(* PLC project mtcs_cover, Institute of Astronomy Onto 0.0.1 *)
(* stored: creationDateTime 2025-01-10T14:32:38.371541, modificationDateTime 2025-01-10T14:32:38.371541 *)

TYPE CoverApertureProcedureStates : (IDLE := 0, ABORTED := 1, PREPARE_PROCESS := 2, ENABLING_RELAYS := 3, ENABLING_MOTORS := 4, ENABLING_MAGNETS := 5, DISABLING_RELAYS := 6, DISABLING_MOTORS := 7, DISABLING_MAGNETS := 8, OPENING_TOP_PANELS := 9, OPENING_BOTH_PANELS := 10, CLOSING_BOTTOM_PANELS := 11, CLOSING_BOTH_PANELS := 12, ERROR := 13, RESETTING := 14, ABORTING := 15);
END_TYPE

TYPE CoverParts : STRUCT
  top : CoverPanelSet;  (* TOP panels *)
  bottom : CoverPanelSet;  (* BOTTOM panels *)
  io : CoverIO;  (* I/O modules *)
  apertureProcedure : CoverApertureProcedure;  (* The closing/opening/... procedure *)
  configManager : ConfigManager;  (* The config manager (to load/save/activate configuration data) *)
END_STRUCT;
END_TYPE

TYPE CoverPanelSetParts : STRUCT
  p1 : CoverPanel;  (* Panel 1 *)
  p2 : CoverPanel;  (* Panel 2 *)
  p3 : CoverPanel;  (* Panel 3 *)
  p4 : CoverPanel;  (* Panel 4 *)
  magnetsRelay : SimpleRelay;  (* Relay for the magnets of this panelset *)
END_STRUCT;
END_TYPE

TYPE CoverPanelParts : STRUCT
  axis : AngularAxis;  (* NC Axis *)
  motorRelay : SimpleRelay;  (* Relay for the motor *)
END_STRUCT;
END_TYPE

TYPE CoverIOParts : STRUCT
  coupler : EtherCatDevice;  (* Coupler *)
  slot1 : EtherCatDevice;  (* Slot 1 *)
  slot2 : EtherCatDevice;  (* Slot 2 *)
  slot3 : EtherCatDevice;  (* Slot 3 *)
  slot4 : EtherCatDevice;  (* Slot 4 *)
  slot5 : EtherCatDevice;  (* Slot 5 *)
  slot6 : EtherCatDevice;  (* Slot 6 *)
  slot7 : EtherCatDevice;  (* Slot 7 *)
  slot8 : EtherCatDevice;  (* Slot 8 *)
  slot9 : EtherCatDevice;  (* Slot 9 *)
  slot10 : EtherCatDevice;  (* Slot 10 *)
  slot11 : EtherCatDevice;  (* Slot 11 *)
  slot12 : EtherCatDevice;  (* Slot 12 *)
  slot13 : EtherCatDevice;  (* Slot 13 *)
END_STRUCT;
END_TYPE

TYPE CoverProcesses : STRUCT
  initialize : Process;  (* Start initializing *)
  lock : Process;  (* Lock the cover *)
  unlock : Process;  (* Unlock the cover *)
  reset : Process;  (* Reset any errors *)
  changeOperatingState : ChangeOperatingStateProcess;  (* Change the operating state (e.g. AUTO, MANUAL, ...) *)
  open : Process;  (* Start opening the cover (only enabled in AUTO mode!) *)
  close : Process;  (* Start closing the cover (only enabled in AUTO mode!) *)
  forceOpen : Process;  (* Start opening the cover EVEN IF WE'RE IN THE UNSAFE REGION *)
  forceClose : Process;  (* Start closing the cover EVEN IF WE'RE IN THE UNSAFE REGION *)
  abort : Process;  (* Abort opening/closing the cover (only enabled in AUTO mode!) *)
END_STRUCT;
END_TYPE

TYPE CoverPanelSetProcesses : STRUCT
  reset : Process;  (* Reset any errors *)
END_STRUCT;
END_TYPE

TYPE CoverPanelProcesses : STRUCT
  startOpening : Process;  (* Start opening the panel *)
  startClosing : Process;  (* Start closing the panel *)
END_STRUCT;
END_TYPE

TYPE CoverStatuses : STRUCT
  initializationStatus : InitializationStatus;
  apertureStatus : ApertureStatus;
  healthStatus : HealthStatus;
  busyStatus : BusyStatus;
  operatingStatus : OperatingStatus;
END_STRUCT;
END_TYPE

TYPE CoverApertureProcedureStatuses : STRUCT
  busyStatus : BusyStatus;  (* Is the CoverApertureProcedure in a busy state? *)
  healthStatus : HealthStatus;  (* Is the CoverApertureProcedure in a healthy state? *)
END_STRUCT;
END_TYPE

TYPE CoverPanelSetStatuses : STRUCT
  apertureStatus : ApertureStatus;
  healthStatus : HealthStatus;
  busyStatus : BusyStatus;
END_STRUCT;
END_TYPE

TYPE CoverPanelStatuses : STRUCT
  busyStatus : BusyStatus;  (* Is the panel in a busy state? *)
  apertureStatus : ApertureStatus;  (* Is the panel open or closed? *)
  healthStatus : HealthStatus;  (* Is the panel in a healthy state? *)
  openingStatus : OpeningStatus;  (* Is the panel opening or closing or standing still? *)
END_STRUCT;
END_TYPE

TYPE CoverIOStatuses : STRUCT
  healthStatus : HealthStatus;  (* Is the I/O in a healthy state? *)
END_STRUCT;
END_TYPE

TYPE CoverConfig : STRUCT
  top : CoverPanelSetConfig;  (* The config of the top panel set *)
  bottom : CoverPanelSetConfig;  (* The config of the bottom panel set *)
  openingVelocity : LREAL := 20.0;  (* The opening velocity of the panels in degrees per second (always positive!) *)
  closingVelocity : LREAL := 20.0;  (* The closing velocity of the panels in degrees per second (always positive!) *)
  magnetRemanentTime : LREAL := 3.0;  (* How many seconds should be waited after disabling a magnet, before a panel may move? *)
  targetDistanceBetweenPanelSets : LREAL;  (* The minimum distance in degrees between both panelsets *)
  minDistanceBetweenPanelSets : LREAL;  (* The minimum distance in degrees between both panelsets *)
  unsafeRangeMinElevation : LREAL;  (* The minimum elevation of the unsafe range *)
  unsafeRangeMinAzimuth : LREAL;  (* The minimum azimuth of the unsafe range *)
  unsafeRangeMaxAzimuth : LREAL;  (* The maximum azimuth of the unsafe range *)
END_STRUCT;
END_TYPE

TYPE CoverPanelSetConfig : STRUCT
  p1 : CoverPanelConfig;  (* The config of the first panel of this set *)
  p2 : CoverPanelConfig;  (* The config of the second panel of this set *)
  p3 : CoverPanelConfig;  (* The config of the third panel of this set *)
  p4 : CoverPanelConfig;  (* The config of the fourth panel of this set *)
  name : STRING;  (* The name of the panel set *)
END_STRUCT;
END_TYPE

TYPE CoverPanelConfig : STRUCT
  closedPosition : LREAL;  (* The closed position of the panel in degrees *)
  openPosition : LREAL;  (* The open position of the panel in degrees *)
  openTolerance : LREAL;  (* The tolerance for opening, in degrees *)
  closedTolerance : LREAL;  (* The tolerance for closing, in degrees *)
  standstillTolerance : LREAL;  (* Tolerance in degrees per second: if smaller than ABS(this value), then the cover panel is considered to be standing still *)
  name : STRING;  (* The name of the panel *)
  offset : LREAL;  (* The offset of the panel w.r.t. north *)
END_STRUCT;
END_TYPE

FUNCTION_BLOCK SM_Cover
  VAR_INPUT
    {attribute 'OPC.UA.DA' := '1'}
    {attribute 'OPC.UA.DA.Access' := '1'}
    editableConfig : CoverConfig;  (* Editable configuration of the cover *)
  END_VAR
  VAR_OUTPUT
    {attribute 'OPC.UA.DA' := '1'}
    {attribute 'OPC.UA.DA.Access' := '1'}
    actualStatus : STRING;  (* Current status description *)
    previousStatus : STRING;  (* Previous status description *)
    {attribute 'OPC.UA.DA' := '1'}
    {attribute 'OPC.UA.DA.Access' := '1'}
    config : CoverConfig;  (* Active configuration of the cover *)
    {attribute 'OPC.UA.DA' := '1'}
    {attribute 'OPC.UA.DA.Access' := '1'}
    currentMeasurement : CurrentMeasurement;  (* The current measurement of the selected panels *)
    {attribute 'OPC.UA.DA' := '1'}
    {attribute 'OPC.UA.DA.Access' := '1'}
    safeToOpenOrClose : BOOL;  (* True if safe to open or close! *)
    statuses : CoverStatuses;  (* Statuses of the state machine *)
    parts : CoverParts;  (* Parts of the state machine *)
    processes : CoverProcesses;  (* Processes of the state machine *)
  END_VAR
  VAR_IN_OUT
    {attribute 'OPC.UA.DA' := '0'}
    operatorStatus : OperatorStatus;
    {attribute 'OPC.UA.DA' := '0'}
    aziPos : AngularPosition;  (* Actual azimuth position of the telescope *)
    {attribute 'OPC.UA.DA' := '0'}
    elePos : AngularPosition;  (* Actual elevation position of the telescope *)
  END_VAR

            currentMeasurement();
parts.top(
    initializationStatus := statuses.initializationStatus,
    operatorStatus := operatorStatus,
    operatingStatus := statuses.operatingStatus,
    config := config.top,
    coverConfig := config);
parts.bottom(
    initializationStatus := statuses.initializationStatus,
    operatorStatus := operatorStatus,
    operatingStatus := statuses.operatingStatus,
    config := config.bottom,
    coverConfig := config);
parts.io();
parts.apertureProcedure(
    top := parts.top,
    bottom := parts.bottom,
    coverConfig := config);
parts.configManager( isEnabled := operatorStatus.tech AND statuses.initializationStatus.initialized );
statuses.initializationStatus();
statuses.apertureStatus(
    isOpen := parts.top.statuses.apertureStatus.open AND parts.bottom.statuses.apertureStatus.open,
    isClosed := parts.top.statuses.apertureStatus.closed AND parts.bottom.statuses.apertureStatus.closed);
statuses.healthStatus(
    isGood := parts.top.statuses.healthStatus.isGood AND (parts.bottom.statuses.healthStatus.isGood AND (parts.apertureProcedure.statuses.healthStatus.isGood AND parts.io.statuses.healthStatus.isGood)),
    hasWarning := (parts.top.statuses.healthStatus.hasWarning OR (parts.bottom.statuses.healthStatus.hasWarning OR (parts.apertureProcedure.statuses.healthStatus.hasWarning OR parts.io.statuses.healthStatus.hasWarning))) OR (statuses.busyStatus.idle AND (NOT(statuses.apertureStatus.open OR statuses.apertureStatus.closed))));
statuses.busyStatus( isBusy := parts.top.statuses.busyStatus.busy OR (parts.bottom.statuses.busyStatus.busy OR parts.apertureProcedure.statuses.busyStatus.busy) );
statuses.operatingStatus( superState := statuses.initializationStatus.initialized );
processes.initialize( isEnabled := statuses.initializationStatus.shutdown OR (statuses.initializationStatus.initializingFailed OR statuses.initializationStatus.initialized) );
processes.lock( isEnabled := operatorStatus.tech AND statuses.initializationStatus.initialized );
processes.unlock( isEnabled := operatorStatus.tech AND statuses.initializationStatus.locked );
processes.reset( isEnabled := (NOT(statuses.initializationStatus.shutdown OR statuses.initializationStatus.locked)) AND (parts.apertureProcedure.state = CoverApertureProcedureStates.ERROR) );
processes.changeOperatingState( isEnabled := statuses.busyStatus.idle AND statuses.initializationStatus.initialized );
processes.open( isEnabled := processes.forceOpen.statuses.enabledStatus.enabled AND safeToOpenOrClose );
processes.close( isEnabled := processes.forceClose.statuses.enabledStatus.enabled AND safeToOpenOrClose );
processes.forceOpen( isEnabled := (statuses.busyStatus.idle OR (statuses.busyStatus.busy AND (parts.apertureProcedure.state = CoverApertureProcedureStates.CLOSING_BOTH_PANELS))) AND (statuses.initializationStatus.initialized AND (statuses.operatingStatus.auto AND (NOT(statuses.apertureStatus.open)))) );
processes.forceClose( isEnabled := (statuses.busyStatus.idle OR (statuses.busyStatus.busy AND (parts.apertureProcedure.state = CoverApertureProcedureStates.OPENING_BOTH_PANELS))) AND (statuses.initializationStatus.initialized AND (statuses.operatingStatus.auto AND (NOT(statuses.apertureStatus.closed)))) );
processes.abort( isEnabled := parts.apertureProcedure.statuses.busyStatus.busy );

          

{attribute 'TcRpcEnable' := '1'}
METHOD initialize : RequestResults
                  initialize := THIS^.processes.initialize.request();

                
END_METHOD

{attribute 'TcRpcEnable' := '1'}
METHOD lock : RequestResults
                  lock := THIS^.processes.lock.request();

                
END_METHOD

{attribute 'TcRpcEnable' := '1'}
METHOD unlock : RequestResults
                  unlock := THIS^.processes.unlock.request();

                
END_METHOD

{attribute 'TcRpcEnable' := '1'}
METHOD reset : RequestResults
                  reset := THIS^.processes.reset.request();

                
END_METHOD

{attribute 'TcRpcEnable' := '1'}
METHOD changeOperatingState : RequestResults
  VAR_INPUT
    state : OperatingStates;
  END_VAR
                  changeOperatingState := THIS^.processes.changeOperatingState.request( state := state );

                
END_METHOD

{attribute 'TcRpcEnable' := '1'}
METHOD open : RequestResults
                  open := THIS^.processes.open.request();

                
END_METHOD

{attribute 'TcRpcEnable' := '1'}
METHOD close : RequestResults
                  close := THIS^.processes.close.request();

                
END_METHOD

{attribute 'TcRpcEnable' := '1'}
METHOD forceOpen : RequestResults
                  forceOpen := THIS^.processes.forceOpen.request();

                
END_METHOD

{attribute 'TcRpcEnable' := '1'}
METHOD forceClose : RequestResults
                  forceClose := THIS^.processes.forceClose.request();

                
END_METHOD

{attribute 'TcRpcEnable' := '1'}
METHOD abort : RequestResults
                  abort := THIS^.processes.abort.request();

                
END_METHOD

{attribute 'TcRpcEnable' := '1'}
METHOD _log : BOOL
  VAR_INPUT
    name : STRING;  (* Name of this function block instance *)
  END_VAR
  VAR_IN_OUT
    buffer : LogBuffer;  (* Buffer to write all logging to *)
  END_VAR
  VAR
    subBuffer : LogBuffer;  (* Temporary buffer to write logging by parts (sub-statemachines) to *)
  END_VAR
                  THIS^.parts.top._log(
    name := 'top',
    buffer := subBuffer);
THIS^.parts.bottom._log(
    name := 'bottom',
    buffer := subBuffer);
THIS^.parts.io._log(
    name := 'io',
    buffer := subBuffer);
THIS^.parts.apertureProcedure._log(
    name := 'apertureProcedure',
    buffer := subBuffer);
THIS^.parts.configManager._log(
    name := 'configManager',
    buffer := subBuffer);
THIS^.processes.initialize._log(
    name := 'processes.initialize',
    buffer := subBuffer);
THIS^.processes.lock._log(
    name := 'processes.lock',
    buffer := subBuffer);
THIS^.processes.unlock._log(
    name := 'processes.unlock',
    buffer := subBuffer);
THIS^.processes.reset._log(
    name := 'processes.reset',
    buffer := subBuffer);
THIS^.processes.changeOperatingState._log(
    name := 'processes.changeOperatingState',
    buffer := subBuffer);
THIS^.processes.open._log(
    name := 'processes.open',
    buffer := subBuffer);
THIS^.processes.close._log(
    name := 'processes.close',
    buffer := subBuffer);
THIS^.processes.forceOpen._log(
    name := 'processes.forceOpen',
    buffer := subBuffer);
THIS^.processes.forceClose._log(
    name := 'processes.forceClose',
    buffer := subBuffer);
THIS^.processes.abort._log(
    name := 'processes.abort',
    buffer := subBuffer);
LOGGER(
    name := name,
    actualStatus := THIS^.actualStatus,
    previousStatus := THIS^.previousStatus,
    buffer := buffer,
    subBuffer := subBuffer,
    pHealthStatus := ADR(THIS^.statuses.healthStatus),
    pBusyStatus := ADR(THIS^.statuses.busyStatus));

                
END_METHOD
END_FUNCTION_BLOCK

FUNCTION_BLOCK SM_CoverApertureProcedure
  VAR_INPUT
    {attribute 'OPC.UA.DA' := '0'}
    state : CoverApertureProcedureStates;  (* New state, to be set by the manual implementation *)
  END_VAR
  VAR_OUTPUT
    {attribute 'OPC.UA.DA' := '1'}
    {attribute 'OPC.UA.DA.Access' := '1'}
    actualStatus : STRING;  (* Current status description *)
    previousStatus : STRING;  (* Previous status description *)
    {attribute 'OPC.UA.DA' := '1'}
    {attribute 'OPC.UA.DA.Access' := '1'}
    opening : BOOL;  (* Is the procedure busy with opening? *)
    {attribute 'OPC.UA.DA' := '1'}
    {attribute 'OPC.UA.DA.Access' := '1'}
    closing : BOOL;  (* Is the procedure busy with closing? *)
    {attribute 'OPC.UA.DA' := '1'}
    {attribute 'OPC.UA.DA.Access' := '1'}
    distance : AngularPosition;  (* The closest distance between the top and bottom panels *)
    statuses : CoverApertureProcedureStatuses;  (* Statuses of the state machine *)
  END_VAR
  VAR_IN_OUT
    {attribute 'OPC.UA.DA' := '0'}
    top : CoverPanelSet;
    {attribute 'OPC.UA.DA' := '0'}
    bottom : CoverPanelSet;
    {attribute 'OPC.UA.DA' := '0'}
    coverConfig : CoverConfig;
  END_VAR

            statuses.busyStatus( isBusy := NOT((state = CoverApertureProcedureStates.IDLE) OR ((state = CoverApertureProcedureStates.ABORTED) OR (state = CoverApertureProcedureStates.ERROR))) );
statuses.healthStatus(
    isGood := NOT(state = CoverApertureProcedureStates.ERROR),
    hasWarning := state = CoverApertureProcedureStates.ABORTED);

          

{attribute 'TcRpcEnable' := '1'}
METHOD _log : BOOL
  VAR_INPUT
    name : STRING;  (* Name of this function block instance *)
  END_VAR
  VAR_IN_OUT
    buffer : LogBuffer;  (* Buffer to write all logging to *)
  END_VAR
  VAR
    subBuffer : LogBuffer;  (* Temporary buffer to write logging by parts (sub-statemachines) to *)
  END_VAR
                  LOGGER(
    name := name,
    actualStatus := THIS^.actualStatus,
    previousStatus := THIS^.previousStatus,
    buffer := buffer,
    subBuffer := subBuffer,
    pHealthStatus := ADR(THIS^.statuses.healthStatus),
    pBusyStatus := ADR(THIS^.statuses.busyStatus));

                
END_METHOD
END_FUNCTION_BLOCK

FUNCTION_BLOCK SM_CoverPanelSet
  VAR_OUTPUT
    {attribute 'OPC.UA.DA' := '1'}
    {attribute 'OPC.UA.DA.Access' := '1'}
    actualStatus : STRING;  (* Current status description *)
    previousStatus : STRING;  (* Previous status description *)
    statuses : CoverPanelSetStatuses;  (* Statuses of the state machine *)
    parts : CoverPanelSetParts;  (* Parts of the state machine *)
    processes : CoverPanelSetProcesses;  (* Processes of the state machine *)
  END_VAR
  VAR_IN_OUT
    {attribute 'OPC.UA.DA' := '0'}
    initializationStatus : InitializationStatus;
    {attribute 'OPC.UA.DA' := '0'}
    operatorStatus : OperatorStatus;
    {attribute 'OPC.UA.DA' := '0'}
    operatingStatus : OperatingStatus;
    {attribute 'OPC.UA.DA' := '0'}
    config : CoverPanelSetConfig;
    {attribute 'OPC.UA.DA' := '0'}
    coverConfig : CoverConfig;
  END_VAR

            parts.p1(
    initializationStatus := initializationStatus,
    operatorStatus := operatorStatus,
    operatingStatus := operatingStatus,
    config := config.p1,
    coverConfig := coverConfig);
parts.p2(
    initializationStatus := initializationStatus,
    operatorStatus := operatorStatus,
    operatingStatus := operatingStatus,
    config := config.p2,
    coverConfig := coverConfig);
parts.p3(
    initializationStatus := initializationStatus,
    operatorStatus := operatorStatus,
    operatingStatus := operatingStatus,
    config := config.p3,
    coverConfig := coverConfig);
parts.p4(
    initializationStatus := initializationStatus,
    operatorStatus := operatorStatus,
    operatingStatus := operatingStatus,
    config := config.p4,
    coverConfig := coverConfig);
parts.magnetsRelay( isEnabled := initializationStatus.initialized AND operatingStatus.manual );
statuses.apertureStatus(
    isOpen := parts.p1.statuses.apertureStatus.open AND (parts.p2.statuses.apertureStatus.open AND (parts.p3.statuses.apertureStatus.open AND parts.p4.statuses.apertureStatus.open)),
    isClosed := parts.p1.statuses.apertureStatus.closed AND (parts.p2.statuses.apertureStatus.closed AND (parts.p3.statuses.apertureStatus.closed AND parts.p4.statuses.apertureStatus.closed)));
statuses.healthStatus(
    isGood := parts.p1.statuses.healthStatus.isGood AND (parts.p2.statuses.healthStatus.isGood AND (parts.p3.statuses.healthStatus.isGood AND parts.p4.statuses.healthStatus.isGood)),
    hasWarning := parts.p1.statuses.healthStatus.hasWarning OR (parts.p2.statuses.healthStatus.hasWarning OR (parts.p3.statuses.healthStatus.hasWarning OR parts.p4.statuses.healthStatus.hasWarning)));
statuses.busyStatus( isBusy := parts.p1.statuses.busyStatus.busy OR (parts.p2.statuses.busyStatus.busy OR (parts.p3.statuses.busyStatus.busy OR parts.p4.statuses.busyStatus.busy)) );
processes.reset( isEnabled := initializationStatus.initialized );

          

{attribute 'TcRpcEnable' := '1'}
METHOD reset : RequestResults
                  reset := THIS^.processes.reset.request();

                
END_METHOD

{attribute 'TcRpcEnable' := '1'}
METHOD _log : BOOL
  VAR_INPUT
    name : STRING;  (* Name of this function block instance *)
  END_VAR
  VAR_IN_OUT
    buffer : LogBuffer;  (* Buffer to write all logging to *)
  END_VAR
  VAR
    subBuffer : LogBuffer;  (* Temporary buffer to write logging by parts (sub-statemachines) to *)
  END_VAR
                  THIS^.parts.p1._log(
    name := 'p1',
    buffer := subBuffer);
THIS^.parts.p2._log(
    name := 'p2',
    buffer := subBuffer);
THIS^.parts.p3._log(
    name := 'p3',
    buffer := subBuffer);
THIS^.parts.p4._log(
    name := 'p4',
    buffer := subBuffer);
THIS^.parts.magnetsRelay._log(
    name := 'magnetsRelay',
    buffer := subBuffer);
THIS^.processes.reset._log(
    name := 'processes.reset',
    buffer := subBuffer);
LOGGER(
    name := name,
    actualStatus := THIS^.actualStatus,
    previousStatus := THIS^.previousStatus,
    buffer := buffer,
    subBuffer := subBuffer,
    pHealthStatus := ADR(THIS^.statuses.healthStatus),
    pBusyStatus := ADR(THIS^.statuses.busyStatus));

                
END_METHOD
END_FUNCTION_BLOCK

FUNCTION_BLOCK SM_CoverPanel
  VAR_INPUT
    {attribute 'OPC.UA.DA' := '1'}
    {attribute 'OPC.UA.DA.Access' := '1'}
    encoderErrorSignal AT %I* : BOOL;  (* Externally read error signal *)
  END_VAR
  VAR_OUTPUT
    {attribute 'OPC.UA.DA' := '1'}
    {attribute 'OPC.UA.DA.Access' := '1'}
    actualStatus : STRING;  (* Current status description *)
    previousStatus : STRING;  (* Previous status description *)
    statuses : CoverPanelStatuses;  (* Statuses of the state machine *)
    parts : CoverPanelParts;  (* Parts of the state machine *)
    processes : CoverPanelProcesses;  (* Processes of the state machine *)
  END_VAR
  VAR_IN_OUT
    {attribute 'OPC.UA.DA' := '0'}
    initializationStatus : InitializationStatus;  (* INITIALIZED or INITIALIZING or ... *)
    {attribute 'OPC.UA.DA' := '0'}
    operatorStatus : OperatorStatus;  (* TECH or OBSERVER or ... *)
    {attribute 'OPC.UA.DA' := '0'}
    operatingStatus : OperatingStatus;  (* MANUAL or AUTO or NONE *)
    {attribute 'OPC.UA.DA' := '0'}
    config : CoverPanelConfig;  (* Configuration of the panel *)
    {attribute 'OPC.UA.DA' := '0'}
    coverConfig : CoverConfig;  (* Configuration of the cover *)
  END_VAR
  VAR
    {attribute 'OPC.UA.DA' := '1'}
    {attribute 'OPC.UA.DA.Access' := '1'}
    encoderErrorSignal_ro : BOOL;
  END_VAR

            parts.axis(
    isEnabled := operatorStatus.tech AND (operatingStatus.manual AND initializationStatus.initialized),
    standstillTolerance := config.standstillTolerance);
parts.motorRelay( isEnabled := parts.axis.isEnabled );
statuses.busyStatus( isBusy := parts.axis.statuses.busyStatus.busy OR parts.motorRelay.statuses.busyStatus.busy );
statuses.apertureStatus(
    isOpen := (ABS(config.openPosition - parts.axis.actPos.degrees.value)) < config.openTolerance,
    isClosed := (ABS(config.closedPosition - parts.axis.actPos.degrees.value)) < config.closedTolerance);
statuses.healthStatus(
    isGood := parts.axis.statuses.healthStatus.isGood AND (NOT(encoderErrorSignal)),
    hasWarning := parts.axis.statuses.healthStatus.hasWarning);
statuses.openingStatus(
    isOpening := parts.axis.statuses.motionStatus.backward,
    isClosing := parts.axis.statuses.motionStatus.forward);
processes.startOpening( isEnabled := operatorStatus.tech AND (operatingStatus.manual AND initializationStatus.initialized) );
processes.startClosing( isEnabled := operatorStatus.tech AND (operatingStatus.manual AND initializationStatus.initialized) );
encoderErrorSignal_ro := encoderErrorSignal;

          

{attribute 'TcRpcEnable' := '1'}
METHOD startOpening : RequestResults
                  startOpening := THIS^.processes.startOpening.request();

                
END_METHOD

{attribute 'TcRpcEnable' := '1'}
METHOD startClosing : RequestResults
                  startClosing := THIS^.processes.startClosing.request();

                
END_METHOD

{attribute 'TcRpcEnable' := '1'}
METHOD _log : BOOL
  VAR_INPUT
    name : STRING;  (* Name of this function block instance *)
  END_VAR
  VAR_IN_OUT
    buffer : LogBuffer;  (* Buffer to write all logging to *)
  END_VAR
  VAR
    subBuffer : LogBuffer;  (* Temporary buffer to write logging by parts (sub-statemachines) to *)
  END_VAR
                  THIS^.parts.axis._log(
    name := 'axis',
    buffer := subBuffer);
THIS^.parts.motorRelay._log(
    name := 'motorRelay',
    buffer := subBuffer);
THIS^.processes.startOpening._log(
    name := 'processes.startOpening',
    buffer := subBuffer);
THIS^.processes.startClosing._log(
    name := 'processes.startClosing',
    buffer := subBuffer);
LOGGER(
    name := name,
    actualStatus := THIS^.actualStatus,
    previousStatus := THIS^.previousStatus,
    buffer := buffer,
    subBuffer := subBuffer,
    pHealthStatus := ADR(THIS^.statuses.healthStatus),
    pBusyStatus := ADR(THIS^.statuses.busyStatus));

                
END_METHOD
END_FUNCTION_BLOCK

FUNCTION_BLOCK SM_CoverIO
  VAR_OUTPUT
    {attribute 'OPC.UA.DA' := '1'}
    {attribute 'OPC.UA.DA.Access' := '1'}
    actualStatus : STRING;  (* Current status description *)
    previousStatus : STRING;  (* Previous status description *)
    statuses : CoverIOStatuses;  (* Statuses of the state machine *)
    parts : CoverIOParts;  (* Parts of the state machine *)
  END_VAR

            parts.coupler(
    id := '110A1',
    typeId := 'EK1101');
parts.slot1(
    id := '115A1',
    typeId := 'EL2008');
parts.slot2(
    id := '116A1',
    typeId := 'EL4008');
parts.slot3(
    id := '117A1',
    typeId := 'EL1088');
parts.slot4(
    id := '118A1',
    typeId := 'EL5002');
parts.slot5(
    id := '118A5',
    typeId := 'EL5002');
parts.slot6(
    id := '119A1',
    typeId := 'EL5002');
parts.slot7(
    id := '119A5',
    typeId := 'EL5002');
parts.slot8(
    id := '111A1',
    typeId := 'EL2622');
parts.slot9(
    id := '111A5',
    typeId := 'EL2622');
parts.slot10(
    id := '112A1',
    typeId := 'EL2622');
parts.slot11(
    id := '112A5',
    typeId := 'EL2622');
parts.slot12(
    id := '113A1',
    typeId := 'EL2622');
parts.slot13(
    id := '114A1',
    typeId := 'EL3681');
statuses.healthStatus( isGood := parts.coupler.statuses.healthStatus.isGood AND (parts.slot1.statuses.healthStatus.isGood AND (parts.slot2.statuses.healthStatus.isGood AND (parts.slot3.statuses.healthStatus.isGood AND (parts.slot4.statuses.healthStatus.isGood AND (parts.slot5.statuses.healthStatus.isGood AND (parts.slot6.statuses.healthStatus.isGood AND (parts.slot7.statuses.healthStatus.isGood AND (parts.slot8.statuses.healthStatus.isGood AND (parts.slot9.statuses.healthStatus.isGood AND (parts.slot10.statuses.healthStatus.isGood AND (parts.slot11.statuses.healthStatus.isGood AND (parts.slot12.statuses.healthStatus.isGood AND parts.slot13.statuses.healthStatus.isGood)))))))))))) );

          

{attribute 'TcRpcEnable' := '1'}
METHOD _log : BOOL
  VAR_INPUT
    name : STRING;  (* Name of this function block instance *)
  END_VAR
  VAR_IN_OUT
    buffer : LogBuffer;  (* Buffer to write all logging to *)
  END_VAR
  VAR
    subBuffer : LogBuffer;  (* Temporary buffer to write logging by parts (sub-statemachines) to *)
  END_VAR
                  THIS^.parts.coupler._log(
    name := 'coupler',
    buffer := subBuffer);
THIS^.parts.slot1._log(
    name := 'slot1',
    buffer := subBuffer);
THIS^.parts.slot2._log(
    name := 'slot2',
    buffer := subBuffer);
THIS^.parts.slot3._log(
    name := 'slot3',
    buffer := subBuffer);
THIS^.parts.slot4._log(
    name := 'slot4',
    buffer := subBuffer);
THIS^.parts.slot5._log(
    name := 'slot5',
    buffer := subBuffer);
THIS^.parts.slot6._log(
    name := 'slot6',
    buffer := subBuffer);
THIS^.parts.slot7._log(
    name := 'slot7',
    buffer := subBuffer);
THIS^.parts.slot8._log(
    name := 'slot8',
    buffer := subBuffer);
THIS^.parts.slot9._log(
    name := 'slot9',
    buffer := subBuffer);
THIS^.parts.slot10._log(
    name := 'slot10',
    buffer := subBuffer);
THIS^.parts.slot11._log(
    name := 'slot11',
    buffer := subBuffer);
THIS^.parts.slot12._log(
    name := 'slot12',
    buffer := subBuffer);
THIS^.parts.slot13._log(
    name := 'slot13',
    buffer := subBuffer);
LOGGER(
    name := name,
    actualStatus := THIS^.actualStatus,
    previousStatus := THIS^.previousStatus,
    buffer := buffer,
    subBuffer := subBuffer,
    pHealthStatus := ADR(THIS^.statuses.healthStatus));

                
END_METHOD
END_FUNCTION_BLOCK
